Omron Sysmac Studio project Proyecto_Analogía (Sysmac Studio 1.23.0.14, StandardProject)

# Controller new_Controller_0: NX1P2-1040DT1 version 1.18
Task PrimaryTask (priority 4, period or condition 2000): Programa0

VAR_GLOBAL
    AI1 : INT;  (* Lectura Analógica 1; at BuiltInIO://opt/#0/Ch1_Analog_Input_Value *)
    AI2 : INT;  (* Lectura Analógica 2; at BuiltInIO://opt/#0/Ch2_Analog_Input_Value *)
    AO1 : INT;  (* Escritura Analógica 1; at BuiltInIO://opt/#0/Ch1_Analog_Output_Value *)
    AO2 : INT;  (* Escritura Analógica 2; at BuiltInIO://opt/#0/Ch2_Analog_Output_Value *)
END_VAR
VAR_GLOBAL RETAIN
    temp1 AT %D10 : REAL;  (* published *)
END_VAR

PROGRAM Programa0
VAR
    var1 : BOOL;
END_VAR
VAR_EXTERNAL
    temp1 : REAL;
    AI1 : INT;
    AO1 : INT;
END_VAR

(* Section Sección0: ladder, written here as Structured Text *)

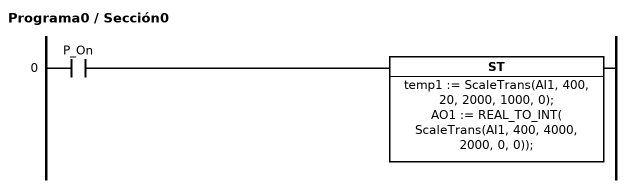
(* Rung 0 *)
IF P_On THEN
    temp1 := ScaleTrans(AI1, 400, 20, 2000, 1000, 0);
    AO1 := REAL_TO_INT(ScaleTrans(AI1, 400, 4000, 2000, 0, 0));
END_IF;
END_PROGRAM